FUNCTION_BLOCK CylinderMaterSlave (* Basic Function Block Type *)
  (* Standard: 61499-2 *)
  (* Version 0.2, 2003-12-04, JHC, Rockwell Automation, Renamed for better indexing. *)
  (* Version 0.1, 2002-11-05, JHC, Rockwell Automation, Corrected missing ST element in Algorithm REQ. *)
  (* Version 0.0, 2000-05-30, JHC, Rockwell Automation *)
  (* Compiler header: package fb.rt.pnp; *)
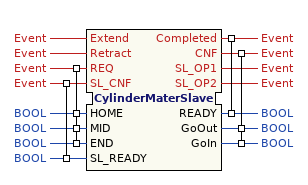
  EVENT_INPUT
    Extend; (* Initialization Request *)
    Retract; (* Normal Execution Request *)
    REQ WITH HOME, MID, END;
    SL_CNF WITH SL_READY;
  END_EVENT
  EVENT_OUTPUT
    Completed WITH READY; (* Initialization Confirm *)
    CNF WITH GoOut, GoIn;
    SL_OP1;
    SL_OP2;
  END_EVENT
  VAR_INPUT
    HOME : BOOL; (* Input event qualifier *)
    MID : BOOL; (* Input event qualifier *)
    END : BOOL; (* Input event qualifier *)
    SL_READY : BOOL;
  END_VAR
  VAR_OUTPUT
    READY : BOOL; (* Output event qualifier *)
    GoOut : BOOL; (* Output event qualifier *)
    GoIn : BOOL; (* Output event qualifier *)
  END_VAR
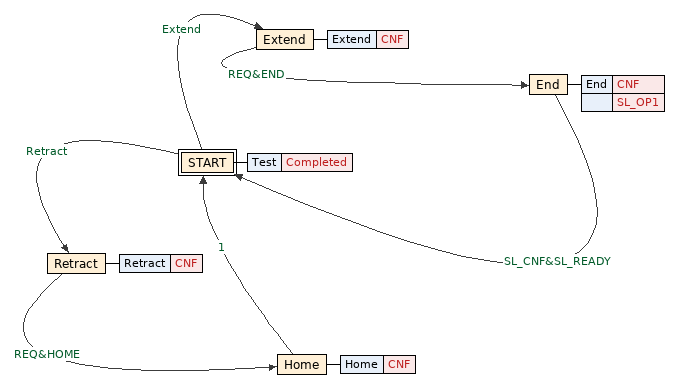
  EC_STATES
    START : Test -> Completed; (* Initial State *)
    Extend : Extend -> CNF; (* Initialization *)
    Retract : Retract -> CNF; (* Normal execution *)
    Home : Home -> CNF; (* Normal execution *)
    End : End -> CNF, -> SL_OP1; (* Normal execution *)
  END_STATES
  EC_TRANSITIONS
    START TO Extend := Extend;
    Extend TO End := REQ&END;
    Retract TO Home := REQ&HOME;
    Home TO START := 1;
    End TO START := SL_CNF&SL_READY;
    START TO Retract := Retract;
  END_TRANSITIONS
  ALGORITHM Extend IN ST: (* Initialization algorithm *)
GoOut := TRUE;
GoIn := FALSE;
READY := FALSE;
System.out.println("ExtendMS!!");
  END_ALGORITHM
  ALGORITHM REQ IN ST: (* Normally executed algorithm *)

  END_ALGORITHM
  ALGORITHM Retract IN ST:
GoIn := TRUE;
GoOut := FALSE;
READY := FALSE;
System.out.println("RetractMS!!");
  END_ALGORITHM
  ALGORITHM Home IN ST:
READY := TRUE;
GoIn := FALSE;
System.out.println("HomeMS!!");
  END_ALGORITHM
  ALGORITHM End IN ST:
READY := TRUE;
GoOut := FALSE;
System.out.println("EndMS!!");
  END_ALGORITHM
  ALGORITHM Wait IN ST:
READY := TRUE;
System.out.println("Wait!!!");
  END_ALGORITHM
  ALGORITHM Test IN ST:
System.out.println("Test");
  END_ALGORITHM
END_FUNCTION_BLOCK
